TYPE ST_MBMStdInput :
STRUCT
    Run_Mode: BIT;  //
END_STRUCT
END_TYPE

(* stored: Version 1.1.0.1, ProductVersion 3.1.4024.12
   DUT ST_MBMStdInput: Id {a602c7fb-7bf3-4067-a5e6-193fab0876f0} *)
